(* IEC 61131-3 sources: TA/Tests/RetainTest/OLD/Structure test (part 9) *)

(* ---- StructureArrayTest.st ---- *)
PROGRAM StructureArrayTest

// СТРУКТУРА МАССИВОВ
IF TRIGGER_IMP.Q THEN

    ARRAY_STRUCTURE_RETAIN.ARRAY_BOOL[0] := NOT ARRAY_STRUCTURE_RETAIN.ARRAY_BOOL[0];
    ARRAY_STRUCTURE_RETAIN.ARRAY_BOOL[1] := NOT ARRAY_STRUCTURE_RETAIN.ARRAY_BOOL[1];
    ARRAY_STRUCTURE_RETAIN.ARRAY_BOOL[2] := NOT ARRAY_STRUCTURE_RETAIN.ARRAY_BOOL[2];
    ARRAY_STRUCTURE_RETAIN.ARRAY_BOOL[3] := NOT ARRAY_STRUCTURE_RETAIN.ARRAY_BOOL[3];
    ARRAY_STRUCTURE_RETAIN.ARRAY_BOOL[4] := NOT ARRAY_STRUCTURE_RETAIN.ARRAY_BOOL[4];
    ARRAY_STRUCTURE_RETAIN.ARRAY_BOOL[5] := NOT ARRAY_STRUCTURE_RETAIN.ARRAY_BOOL[5];
    ARRAY_STRUCTURE_RETAIN.ARRAY_BOOL[6] := NOT ARRAY_STRUCTURE_RETAIN.ARRAY_BOOL[6];
    ARRAY_STRUCTURE_RETAIN.ARRAY_BOOL[7] := NOT ARRAY_STRUCTURE_RETAIN.ARRAY_BOOL[7];
    ARRAY_STRUCTURE_RETAIN.ARRAY_BOOL[8] := ARRAY_STRUCTURE_RETAIN.ARRAY_BOOL[6];
    ARRAY_STRUCTURE_RETAIN.ARRAY_BOOL[9] := ARRAY_STRUCTURE_RETAIN.ARRAY_BOOL[7];

    ARRAY_STRUCTURE_RETAIN.ARRAY_BYTE[0] := ARRAY_STRUCTURE_RETAIN.ARRAY_BYTE[0] + 1;
    ARRAY_STRUCTURE_RETAIN.ARRAY_BYTE[1] := ARRAY_STRUCTURE_RETAIN.ARRAY_BYTE[1] + 1;
    ARRAY_STRUCTURE_RETAIN.ARRAY_BYTE[2] := ARRAY_STRUCTURE_RETAIN.ARRAY_BYTE[2] + 1;
    ARRAY_STRUCTURE_RETAIN.ARRAY_BYTE[3] := ARRAY_STRUCTURE_RETAIN.ARRAY_BYTE[3] + 1;
    ARRAY_STRUCTURE_RETAIN.ARRAY_BYTE[4] := ARRAY_STRUCTURE_RETAIN.ARRAY_BYTE[4] + 1;
    ARRAY_STRUCTURE_RETAIN.ARRAY_BYTE[5] := ARRAY_STRUCTURE_RETAIN.ARRAY_BYTE[5] + 1;
    ARRAY_STRUCTURE_RETAIN.ARRAY_BYTE[6] := ARRAY_STRUCTURE_RETAIN.ARRAY_BYTE[6] + 1;
    ARRAY_STRUCTURE_RETAIN.ARRAY_BYTE[7] := ARRAY_STRUCTURE_RETAIN.ARRAY_BYTE[7] + 1;
    ARRAY_STRUCTURE_RETAIN.ARRAY_BYTE[8] := ARRAY_STRUCTURE_RETAIN.ARRAY_BYTE[6];
    ARRAY_STRUCTURE_RETAIN.ARRAY_BYTE[9] := ARRAY_STRUCTURE_RETAIN.ARRAY_BYTE[7];

    ARRAY_STRUCTURE_RETAIN.ARRAY_DATE[0] := ANY_TO_DATE(1445385600 + ARRAY_STRUCTURE_RETAIN.ARRAY_DINT[0] * 86400);
    ARRAY_STRUCTURE_RETAIN.ARRAY_DATE[1] := ANY_TO_DATE(1445385600 + ARRAY_STRUCTURE_RETAIN.ARRAY_DINT[1] * 86400);
    ARRAY_STRUCTURE_RETAIN.ARRAY_DATE[2] := ANY_TO_DATE(1445385600 + ARRAY_STRUCTURE_RETAIN.ARRAY_DINT[2] * 86400);
    ARRAY_STRUCTURE_RETAIN.ARRAY_DATE[3] := ANY_TO_DATE(1445385600 + ARRAY_STRUCTURE_RETAIN.ARRAY_DINT[3] * 86400);
    ARRAY_STRUCTURE_RETAIN.ARRAY_DATE[4] := ANY_TO_DATE(1445385600 + ARRAY_STRUCTURE_RETAIN.ARRAY_DINT[4] * 86400);
    ARRAY_STRUCTURE_RETAIN.ARRAY_DATE[5] := ANY_TO_DATE(1445385600 + ARRAY_STRUCTURE_RETAIN.ARRAY_DINT[5] * 86400);
    ARRAY_STRUCTURE_RETAIN.ARRAY_DATE[6] := ANY_TO_DATE(1445385600 + ARRAY_STRUCTURE_RETAIN.ARRAY_DINT[6] * 86400);
    ARRAY_STRUCTURE_RETAIN.ARRAY_DATE[7] := ANY_TO_DATE(1445385600 + ARRAY_STRUCTURE_RETAIN.ARRAY_DINT[7] * 86400);
    ARRAY_STRUCTURE_RETAIN.ARRAY_DATE[8] := ARRAY_STRUCTURE_RETAIN.ARRAY_DATE[6];
    ARRAY_STRUCTURE_RETAIN.ARRAY_DATE[9] := ARRAY_STRUCTURE_RETAIN.ARRAY_DATE[7];

    ARRAY_STRUCTURE_RETAIN.ARRAY_DINT[0] := ARRAY_STRUCTURE_RETAIN.ARRAY_DINT[0] + 1;
    ARRAY_STRUCTURE_RETAIN.ARRAY_DINT[1] := ARRAY_STRUCTURE_RETAIN.ARRAY_DINT[1] + 1;
    ARRAY_STRUCTURE_RETAIN.ARRAY_DINT[2] := ARRAY_STRUCTURE_RETAIN.ARRAY_DINT[2] + 1;
    ARRAY_STRUCTURE_RETAIN.ARRAY_DINT[3] := ARRAY_STRUCTURE_RETAIN.ARRAY_DINT[3] + 1;
    ARRAY_STRUCTURE_RETAIN.ARRAY_DINT[4] := ARRAY_STRUCTURE_RETAIN.ARRAY_DINT[4] + 1;
    ARRAY_STRUCTURE_RETAIN.ARRAY_DINT[5] := ARRAY_STRUCTURE_RETAIN.ARRAY_DINT[5] + 1;
    ARRAY_STRUCTURE_RETAIN.ARRAY_DINT[6] := ARRAY_STRUCTURE_RETAIN.ARRAY_DINT[6] + 1;
    ARRAY_STRUCTURE_RETAIN.ARRAY_DINT[7] := ARRAY_STRUCTURE_RETAIN.ARRAY_DINT[7] + 1;
    ARRAY_STRUCTURE_RETAIN.ARRAY_DINT[8] := ARRAY_STRUCTURE_RETAIN.ARRAY_DINT[6];
    ARRAY_STRUCTURE_RETAIN.ARRAY_DINT[9] := ARRAY_STRUCTURE_RETAIN.ARRAY_DINT[7];

    ARRAY_STRUCTURE_RETAIN.ARRAY_DWORD[0] := ARRAY_STRUCTURE_RETAIN.ARRAY_DWORD[0] + 1;
    ARRAY_STRUCTURE_RETAIN.ARRAY_DWORD[1] := ARRAY_STRUCTURE_RETAIN.ARRAY_DWORD[1] + 1;
    ARRAY_STRUCTURE_RETAIN.ARRAY_DWORD[2] := ARRAY_STRUCTURE_RETAIN.ARRAY_DWORD[2] + 1;
    ARRAY_STRUCTURE_RETAIN.ARRAY_DWORD[3] := ARRAY_STRUCTURE_RETAIN.ARRAY_DWORD[3] + 1;
    ARRAY_STRUCTURE_RETAIN.ARRAY_DWORD[4] := ARRAY_STRUCTURE_RETAIN.ARRAY_DWORD[4] + 1;
    ARRAY_STRUCTURE_RETAIN.ARRAY_DWORD[5] := ARRAY_STRUCTURE_RETAIN.ARRAY_DWORD[5] + 1;
    ARRAY_STRUCTURE_RETAIN.ARRAY_DWORD[6] := ARRAY_STRUCTURE_RETAIN.ARRAY_DWORD[6] + 1;
    ARRAY_STRUCTURE_RETAIN.ARRAY_DWORD[7] := ARRAY_STRUCTURE_RETAIN.ARRAY_DWORD[7] + 1;
    ARRAY_STRUCTURE_RETAIN.ARRAY_DWORD[8] := ARRAY_STRUCTURE_RETAIN.ARRAY_DWORD[6];
    ARRAY_STRUCTURE_RETAIN.ARRAY_DWORD[9] := ARRAY_STRUCTURE_RETAIN.ARRAY_DWORD[7];

    ARRAY_STRUCTURE_RETAIN.ARRAY_INT[0] := ARRAY_STRUCTURE_RETAIN.ARRAY_INT[0] + 1;
    ARRAY_STRUCTURE_RETAIN.ARRAY_INT[1] := ARRAY_STRUCTURE_RETAIN.ARRAY_INT[1] + 1;
    ARRAY_STRUCTURE_RETAIN.ARRAY_INT[2] := ARRAY_STRUCTURE_RETAIN.ARRAY_INT[2] + 1;
    ARRAY_STRUCTURE_RETAIN.ARRAY_INT[3] := ARRAY_STRUCTURE_RETAIN.ARRAY_INT[3] + 1;
    ARRAY_STRUCTURE_RETAIN.ARRAY_INT[4] := ARRAY_STRUCTURE_RETAIN.ARRAY_INT[4] + 1;
    ARRAY_STRUCTURE_RETAIN.ARRAY_INT[5] := ARRAY_STRUCTURE_RETAIN.ARRAY_INT[5] + 1;
    ARRAY_STRUCTURE_RETAIN.ARRAY_INT[6] := ARRAY_STRUCTURE_RETAIN.ARRAY_INT[6] + 1;
    ARRAY_STRUCTURE_RETAIN.ARRAY_INT[7] := ARRAY_STRUCTURE_RETAIN.ARRAY_INT[7] + 1;
    ARRAY_STRUCTURE_RETAIN.ARRAY_INT[8] := ARRAY_STRUCTURE_RETAIN.ARRAY_INT[6];
    ARRAY_STRUCTURE_RETAIN.ARRAY_INT[9] := ARRAY_STRUCTURE_RETAIN.ARRAY_INT[7];

    ARRAY_STRUCTURE_RETAIN.ARRAY_LINT[0] := ARRAY_STRUCTURE_RETAIN.ARRAY_LINT[0] + 1;
    ARRAY_STRUCTURE_RETAIN.ARRAY_LINT[1] := ARRAY_STRUCTURE_RETAIN.ARRAY_LINT[1] + 1;
    ARRAY_STRUCTURE_RETAIN.ARRAY_LINT[2] := ARRAY_STRUCTURE_RETAIN.ARRAY_LINT[2] + 1;
    ARRAY_STRUCTURE_RETAIN.ARRAY_LINT[3] := ARRAY_STRUCTURE_RETAIN.ARRAY_LINT[3] + 1;
    ARRAY_STRUCTURE_RETAIN.ARRAY_LINT[4] := ARRAY_STRUCTURE_RETAIN.ARRAY_LINT[4] + 1;
    ARRAY_STRUCTURE_RETAIN.ARRAY_LINT[5] := ARRAY_STRUCTURE_RETAIN.ARRAY_LINT[5] + 1;
    ARRAY_STRUCTURE_RETAIN.ARRAY_LINT[6] := ARRAY_STRUCTURE_RETAIN.ARRAY_LINT[6] + 1;
    ARRAY_STRUCTURE_RETAIN.ARRAY_LINT[7] := ARRAY_STRUCTURE_RETAIN.ARRAY_LINT[7] + 1;
    ARRAY_STRUCTURE_RETAIN.ARRAY_LINT[8] := ARRAY_STRUCTURE_RETAIN.ARRAY_LINT[6];
    ARRAY_STRUCTURE_RETAIN.ARRAY_LINT[9] := ARRAY_STRUCTURE_RETAIN.ARRAY_LINT[7];

    ARRAY_STRUCTURE_RETAIN.ARRAY_LREAL[0] := ARRAY_STRUCTURE_RETAIN.ARRAY_LREAL[0] + 1;
    ARRAY_STRUCTURE_RETAIN.ARRAY_LREAL[1] := ARRAY_STRUCTURE_RETAIN.ARRAY_LREAL[1] + 1;
    ARRAY_STRUCTURE_RETAIN.ARRAY_LREAL[2] := ARRAY_STRUCTURE_RETAIN.ARRAY_LREAL[2] + 1;
    ARRAY_STRUCTURE_RETAIN.ARRAY_LREAL[3] := ARRAY_STRUCTURE_RETAIN.ARRAY_LREAL[3] + 1;
    ARRAY_STRUCTURE_RETAIN.ARRAY_LREAL[4] := ARRAY_STRUCTURE_RETAIN.ARRAY_LREAL[4] + 1;
    ARRAY_STRUCTURE_RETAIN.ARRAY_LREAL[5] := ARRAY_STRUCTURE_RETAIN.ARRAY_LREAL[5] + 1;
    ARRAY_STRUCTURE_RETAIN.ARRAY_LREAL[6] := ARRAY_STRUCTURE_RETAIN.ARRAY_LREAL[6] + 1;
    ARRAY_STRUCTURE_RETAIN.ARRAY_LREAL[7] := ARRAY_STRUCTURE_RETAIN.ARRAY_LREAL[7] + 1;
    ARRAY_STRUCTURE_RETAIN.ARRAY_LREAL[8] := ARRAY_STRUCTURE_RETAIN.ARRAY_LREAL[6];
    ARRAY_STRUCTURE_RETAIN.ARRAY_LREAL[9] := ARRAY_STRUCTURE_RETAIN.ARRAY_LREAL[7];

    ARRAY_STRUCTURE_RETAIN.ARRAY_LWORD[0] := ARRAY_STRUCTURE_RETAIN.ARRAY_LWORD[0] + 1;
    ARRAY_STRUCTURE_RETAIN.ARRAY_LWORD[1] := ARRAY_STRUCTURE_RETAIN.ARRAY_LWORD[1] + 1;
    ARRAY_STRUCTURE_RETAIN.ARRAY_LWORD[2] := ARRAY_STRUCTURE_RETAIN.ARRAY_LWORD[2] + 1;
    ARRAY_STRUCTURE_RETAIN.ARRAY_LWORD[3] := ARRAY_STRUCTURE_RETAIN.ARRAY_LWORD[3] + 1;
    ARRAY_STRUCTURE_RETAIN.ARRAY_LWORD[4] := ARRAY_STRUCTURE_RETAIN.ARRAY_LWORD[4] + 1;
    ARRAY_STRUCTURE_RETAIN.ARRAY_LWORD[5] := ARRAY_STRUCTURE_RETAIN.ARRAY_LWORD[5] + 1;
    ARRAY_STRUCTURE_RETAIN.ARRAY_LWORD[6] := ARRAY_STRUCTURE_RETAIN.ARRAY_LWORD[6] + 1;
    ARRAY_STRUCTURE_RETAIN.ARRAY_LWORD[7] := ARRAY_STRUCTURE_RETAIN.ARRAY_LWORD[7] + 1;
    ARRAY_STRUCTURE_RETAIN.ARRAY_LWORD[8] := ARRAY_STRUCTURE_RETAIN.ARRAY_LWORD[6];
    ARRAY_STRUCTURE_RETAIN.ARRAY_LWORD[9] := ARRAY_STRUCTURE_RETAIN.ARRAY_LWORD[7];

    ARRAY_STRUCTURE_RETAIN.ARRAY_REAL[0] := ARRAY_STRUCTURE_RETAIN.ARRAY_REAL[0] + 1;
    ARRAY_STRUCTURE_RETAIN.ARRAY_REAL[1] := ARRAY_STRUCTURE_RETAIN.ARRAY_REAL[1] + 1;
    ARRAY_STRUCTURE_RETAIN.ARRAY_REAL[2] := ARRAY_STRUCTURE_RETAIN.ARRAY_REAL[2] + 1;
    ARRAY_STRUCTURE_RETAIN.ARRAY_REAL[3] := ARRAY_STRUCTURE_RETAIN.ARRAY_REAL[3] + 1;
    ARRAY_STRUCTURE_RETAIN.ARRAY_REAL[4] := ARRAY_STRUCTURE_RETAIN.ARRAY_REAL[4] + 1;
    ARRAY_STRUCTURE_RETAIN.ARRAY_REAL[5] := ARRAY_STRUCTURE_RETAIN.ARRAY_REAL[5] + 1;
    ARRAY_STRUCTURE_RETAIN.ARRAY_REAL[6] := ARRAY_STRUCTURE_RETAIN.ARRAY_REAL[6] + 1;
    ARRAY_STRUCTURE_RETAIN.ARRAY_REAL[7] := ARRAY_STRUCTURE_RETAIN.ARRAY_REAL[7] + 1;
    ARRAY_STRUCTURE_RETAIN.ARRAY_REAL[8] := ARRAY_STRUCTURE_RETAIN.ARRAY_REAL[6];
    ARRAY_STRUCTURE_RETAIN.ARRAY_REAL[9] := ARRAY_STRUCTURE_RETAIN.ARRAY_REAL[7];

    ARRAY_STRUCTURE_RETAIN.ARRAY_SINT[0] := ARRAY_STRUCTURE_RETAIN.ARRAY_SINT[0] + 1;
    ARRAY_STRUCTURE_RETAIN.ARRAY_SINT[1] := ARRAY_STRUCTURE_RETAIN.ARRAY_SINT[1] + 1;
    ARRAY_STRUCTURE_RETAIN.ARRAY_SINT[2] := ARRAY_STRUCTURE_RETAIN.ARRAY_SINT[2] + 1;
    ARRAY_STRUCTURE_RETAIN.ARRAY_SINT[3] := ARRAY_STRUCTURE_RETAIN.ARRAY_SINT[3] + 1;
    ARRAY_STRUCTURE_RETAIN.ARRAY_SINT[4] := ARRAY_STRUCTURE_RETAIN.ARRAY_SINT[4] + 1;
    ARRAY_STRUCTURE_RETAIN.ARRAY_SINT[5] := ARRAY_STRUCTURE_RETAIN.ARRAY_SINT[5] + 1;
    ARRAY_STRUCTURE_RETAIN.ARRAY_SINT[6] := ARRAY_STRUCTURE_RETAIN.ARRAY_SINT[6] + 1;
    ARRAY_STRUCTURE_RETAIN.ARRAY_SINT[7] := ARRAY_STRUCTURE_RETAIN.ARRAY_SINT[7] + 1;
    ARRAY_STRUCTURE_RETAIN.ARRAY_SINT[8] := ARRAY_STRUCTURE_RETAIN.ARRAY_SINT[6];
    ARRAY_STRUCTURE_RETAIN.ARRAY_SINT[9] := ARRAY_STRUCTURE_RETAIN.ARRAY_SINT[7];

    ARRAY_STRUCTURE_RETAIN.ARRAY_STRING[0] := ANY_TO_STRING(ARRAY_STRUCTURE_RETAIN.ARRAY_DINT[0]) + ' ' + ANY_TO_STRING(ARRAY_STRUCTURE_RETAIN.ARRAY_TIME[0]);
    ARRAY_STRUCTURE_RETAIN.ARRAY_STRING[1] := ANY_TO_STRING(ARRAY_STRUCTURE_RETAIN.ARRAY_DINT[1]) + ' ' + ANY_TO_STRING(ARRAY_STRUCTURE_RETAIN.ARRAY_TIME[1]);
    ARRAY_STRUCTURE_RETAIN.ARRAY_STRING[2] := ANY_TO_STRING(ARRAY_STRUCTURE_RETAIN.ARRAY_DINT[2]) + ' ' + ANY_TO_STRING(ARRAY_STRUCTURE_RETAIN.ARRAY_TIME[2]);
    ARRAY_STRUCTURE_RETAIN.ARRAY_STRING[3] := ANY_TO_STRING(ARRAY_STRUCTURE_RETAIN.ARRAY_DINT[3]) + ' ' + ANY_TO_STRING(ARRAY_STRUCTURE_RETAIN.ARRAY_TIME[3]);
    ARRAY_STRUCTURE_RETAIN.ARRAY_STRING[4] := ANY_TO_STRING(ARRAY_STRUCTURE_RETAIN.ARRAY_DINT[4]) + ' ' + ANY_TO_STRING(ARRAY_STRUCTURE_RETAIN.ARRAY_TIME[4]);
    ARRAY_STRUCTURE_RETAIN.ARRAY_STRING[5] := ANY_TO_STRING(ARRAY_STRUCTURE_RETAIN.ARRAY_DINT[5]) + ' ' + ANY_TO_STRING(ARRAY_STRUCTURE_RETAIN.ARRAY_TIME[5]);
    ARRAY_STRUCTURE_RETAIN.ARRAY_STRING[6] := ANY_TO_STRING(ARRAY_STRUCTURE_RETAIN.ARRAY_DINT[6]) + ' ' + ANY_TO_STRING(ARRAY_STRUCTURE_RETAIN.ARRAY_TIME[6]);
    ARRAY_STRUCTURE_RETAIN.ARRAY_STRING[7] := ANY_TO_STRING(ARRAY_STRUCTURE_RETAIN.ARRAY_DINT[7]) + ' ' + ANY_TO_STRING(ARRAY_STRUCTURE_RETAIN.ARRAY_TIME[7]);
    ARRAY_STRUCTURE_RETAIN.ARRAY_STRING[8] := ARRAY_STRUCTURE_RETAIN.ARRAY_STRING[6];
    ARRAY_STRUCTURE_RETAIN.ARRAY_STRING[9] := ARRAY_STRUCTURE_RETAIN.ARRAY_STRING[7];

    ARRAY_STRUCTURE_RETAIN.ARRAY_TIME[0] := ARRAY_STRUCTURE_RETAIN.ARRAY_TIME[0] + PULSE_TIME;
    ARRAY_STRUCTURE_RETAIN.ARRAY_TIME[1] := ARRAY_STRUCTURE_RETAIN.ARRAY_TIME[1] + PULSE_TIME;
    ARRAY_STRUCTURE_RETAIN.ARRAY_TIME[2] := ARRAY_STRUCTURE_RETAIN.ARRAY_TIME[2] + PULSE_TIME;
    ARRAY_STRUCTURE_RETAIN.ARRAY_TIME[3] := ARRAY_STRUCTURE_RETAIN.ARRAY_TIME[3] + PULSE_TIME;
    ARRAY_STRUCTURE_RETAIN.ARRAY_TIME[4] := ARRAY_STRUCTURE_RETAIN.ARRAY_TIME[4] + PULSE_TIME;
    ARRAY_STRUCTURE_RETAIN.ARRAY_TIME[5] := ARRAY_STRUCTURE_RETAIN.ARRAY_TIME[5] + PULSE_TIME;
    ARRAY_STRUCTURE_RETAIN.ARRAY_TIME[6] := ARRAY_STRUCTURE_RETAIN.ARRAY_TIME[6] + PULSE_TIME;
    ARRAY_STRUCTURE_RETAIN.ARRAY_TIME[7] := ARRAY_STRUCTURE_RETAIN.ARRAY_TIME[7] + PULSE_TIME;
    ARRAY_STRUCTURE_RETAIN.ARRAY_TIME[8] := ARRAY_STRUCTURE_RETAIN.ARRAY_TIME[6];
    ARRAY_STRUCTURE_RETAIN.ARRAY_TIME[9] := ARRAY_STRUCTURE_RETAIN.ARRAY_TIME[7];

    ARRAY_STRUCTURE_RETAIN.ARRAY_UDINT[0] := ARRAY_STRUCTURE_RETAIN.ARRAY_UDINT[0] + 1;
    ARRAY_STRUCTURE_RETAIN.ARRAY_UDINT[1] := ARRAY_STRUCTURE_RETAIN.ARRAY_UDINT[1] + 1;
    ARRAY_STRUCTURE_RETAIN.ARRAY_UDINT[2] := ARRAY_STRUCTURE_RETAIN.ARRAY_UDINT[2] + 1;
    ARRAY_STRUCTURE_RETAIN.ARRAY_UDINT[3] := ARRAY_STRUCTURE_RETAIN.ARRAY_UDINT[3] + 1;
    ARRAY_STRUCTURE_RETAIN.ARRAY_UDINT[4] := ARRAY_STRUCTURE_RETAIN.ARRAY_UDINT[4] + 1;
    ARRAY_STRUCTURE_RETAIN.ARRAY_UDINT[5] := ARRAY_STRUCTURE_RETAIN.ARRAY_UDINT[5] + 1;
    ARRAY_STRUCTURE_RETAIN.ARRAY_UDINT[6] := ARRAY_STRUCTURE_RETAIN.ARRAY_UDINT[6] + 1;
    ARRAY_STRUCTURE_RETAIN.ARRAY_UDINT[7] := ARRAY_STRUCTURE_RETAIN.ARRAY_UDINT[7] + 1;
    ARRAY_STRUCTURE_RETAIN.ARRAY_UDINT[8] := ARRAY_STRUCTURE_RETAIN.ARRAY_UDINT[6];
    ARRAY_STRUCTURE_RETAIN.ARRAY_UDINT[9] := ARRAY_STRUCTURE_RETAIN.ARRAY_UDINT[7];

    ARRAY_STRUCTURE_RETAIN.ARRAY_UINT[0] := ARRAY_STRUCTURE_RETAIN.ARRAY_UINT[0] + 1;
    ARRAY_STRUCTURE_RETAIN.ARRAY_UINT[1] := ARRAY_STRUCTURE_RETAIN.ARRAY_UINT[1] + 1;
    ARRAY_STRUCTURE_RETAIN.ARRAY_UINT[2] := ARRAY_STRUCTURE_RETAIN.ARRAY_UINT[2] + 1;
    ARRAY_STRUCTURE_RETAIN.ARRAY_UINT[3] := ARRAY_STRUCTURE_RETAIN.ARRAY_UINT[3] + 1;
    ARRAY_STRUCTURE_RETAIN.ARRAY_UINT[4] := ARRAY_STRUCTURE_RETAIN.ARRAY_UINT[4] + 1;
    ARRAY_STRUCTURE_RETAIN.ARRAY_UINT[5] := ARRAY_STRUCTURE_RETAIN.ARRAY_UINT[5] + 1;
    ARRAY_STRUCTURE_RETAIN.ARRAY_UINT[6] := ARRAY_STRUCTURE_RETAIN.ARRAY_UINT[6] + 1;
    ARRAY_STRUCTURE_RETAIN.ARRAY_UINT[7] := ARRAY_STRUCTURE_RETAIN.ARRAY_UINT[7] + 1;
    ARRAY_STRUCTURE_RETAIN.ARRAY_UINT[8] := ARRAY_STRUCTURE_RETAIN.ARRAY_UINT[6];
    ARRAY_STRUCTURE_RETAIN.ARRAY_UINT[9] := ARRAY_STRUCTURE_RETAIN.ARRAY_UINT[7];

    ARRAY_STRUCTURE_RETAIN.ARRAY_ULINT[0] := ARRAY_STRUCTURE_RETAIN.ARRAY_ULINT[0] + 1;
    ARRAY_STRUCTURE_RETAIN.ARRAY_ULINT[1] := ARRAY_STRUCTURE_RETAIN.ARRAY_ULINT[1] + 1;
    ARRAY_STRUCTURE_RETAIN.ARRAY_ULINT[2] := ARRAY_STRUCTURE_RETAIN.ARRAY_ULINT[2] + 1;
    ARRAY_STRUCTURE_RETAIN.ARRAY_ULINT[3] := ARRAY_STRUCTURE_RETAIN.ARRAY_ULINT[3] + 1;
    ARRAY_STRUCTURE_RETAIN.ARRAY_ULINT[4] := ARRAY_STRUCTURE_RETAIN.ARRAY_ULINT[4] + 1;
    ARRAY_STRUCTURE_RETAIN.ARRAY_ULINT[5] := ARRAY_STRUCTURE_RETAIN.ARRAY_ULINT[5] + 1;
    ARRAY_STRUCTURE_RETAIN.ARRAY_ULINT[6] := ARRAY_STRUCTURE_RETAIN.ARRAY_ULINT[6] + 1;
    ARRAY_STRUCTURE_RETAIN.ARRAY_ULINT[7] := ARRAY_STRUCTURE_RETAIN.ARRAY_ULINT[7] + 1;
    ARRAY_STRUCTURE_RETAIN.ARRAY_ULINT[8] := ARRAY_STRUCTURE_RETAIN.ARRAY_ULINT[6];
    ARRAY_STRUCTURE_RETAIN.ARRAY_ULINT[9] := ARRAY_STRUCTURE_RETAIN.ARRAY_ULINT[7];

    ARRAY_STRUCTURE_RETAIN.ARRAY_USINT[0] := ARRAY_STRUCTURE_RETAIN.ARRAY_USINT[0] + 1;
    ARRAY_STRUCTURE_RETAIN.ARRAY_USINT[1] := ARRAY_STRUCTURE_RETAIN.ARRAY_USINT[1] + 1;
    ARRAY_STRUCTURE_RETAIN.ARRAY_USINT[2] := ARRAY_STRUCTURE_RETAIN.ARRAY_USINT[2] + 1;
    ARRAY_STRUCTURE_RETAIN.ARRAY_USINT[3] := ARRAY_STRUCTURE_RETAIN.ARRAY_USINT[3] + 1;
    ARRAY_STRUCTURE_RETAIN.ARRAY_USINT[4] := ARRAY_STRUCTURE_RETAIN.ARRAY_USINT[4] + 1;
    ARRAY_STRUCTURE_RETAIN.ARRAY_USINT[5] := ARRAY_STRUCTURE_RETAIN.ARRAY_USINT[5] + 1;
    ARRAY_STRUCTURE_RETAIN.ARRAY_USINT[6] := ARRAY_STRUCTURE_RETAIN.ARRAY_USINT[6] + 1;
    ARRAY_STRUCTURE_RETAIN.ARRAY_USINT[7] := ARRAY_STRUCTURE_RETAIN.ARRAY_USINT[7] + 1;
    ARRAY_STRUCTURE_RETAIN.ARRAY_USINT[8] := ARRAY_STRUCTURE_RETAIN.ARRAY_USINT[6];
    ARRAY_STRUCTURE_RETAIN.ARRAY_USINT[9] := ARRAY_STRUCTURE_RETAIN.ARRAY_USINT[7];

    ARRAY_STRUCTURE_RETAIN.ARRAY_WORD[0] := ARRAY_STRUCTURE_RETAIN.ARRAY_WORD[0] + 1;
    ARRAY_STRUCTURE_RETAIN.ARRAY_WORD[1] := ARRAY_STRUCTURE_RETAIN.ARRAY_WORD[1] + 1;
    ARRAY_STRUCTURE_RETAIN.ARRAY_WORD[2] := ARRAY_STRUCTURE_RETAIN.ARRAY_WORD[2] + 1;
    ARRAY_STRUCTURE_RETAIN.ARRAY_WORD[3] := ARRAY_STRUCTURE_RETAIN.ARRAY_WORD[3] + 1;
    ARRAY_STRUCTURE_RETAIN.ARRAY_WORD[4] := ARRAY_STRUCTURE_RETAIN.ARRAY_WORD[4] + 1;
    ARRAY_STRUCTURE_RETAIN.ARRAY_WORD[5] := ARRAY_STRUCTURE_RETAIN.ARRAY_WORD[5] + 1;
    ARRAY_STRUCTURE_RETAIN.ARRAY_WORD[6] := ARRAY_STRUCTURE_RETAIN.ARRAY_WORD[6] + 1;
    ARRAY_STRUCTURE_RETAIN.ARRAY_WORD[7] := ARRAY_STRUCTURE_RETAIN.ARRAY_WORD[7] + 1;
    ARRAY_STRUCTURE_RETAIN.ARRAY_WORD[8] := ARRAY_STRUCTURE_RETAIN.ARRAY_WORD[6];
    ARRAY_STRUCTURE_RETAIN.ARRAY_WORD[9] := ARRAY_STRUCTURE_RETAIN.ARRAY_WORD[7];

    ARRAY_STRUCTURE_NON_RETAIN.ARRAY_BOOL[0] := NOT ARRAY_STRUCTURE_NON_RETAIN.ARRAY_BOOL[0];
    ARRAY_STRUCTURE_NON_RETAIN.ARRAY_BOOL[1] := NOT ARRAY_STRUCTURE_NON_RETAIN.ARRAY_BOOL[1];
    ARRAY_STRUCTURE_NON_RETAIN.ARRAY_BOOL[2] := NOT ARRAY_STRUCTURE_NON_RETAIN.ARRAY_BOOL[2];
    ARRAY_STRUCTURE_NON_RETAIN.ARRAY_BOOL[3] := NOT ARRAY_STRUCTURE_NON_RETAIN.ARRAY_BOOL[3];
    ARRAY_STRUCTURE_NON_RETAIN.ARRAY_BOOL[4] := NOT ARRAY_STRUCTURE_NON_RETAIN.ARRAY_BOOL[4];
    ARRAY_STRUCTURE_NON_RETAIN.ARRAY_BOOL[5] := NOT ARRAY_STRUCTURE_NON_RETAIN.ARRAY_BOOL[5];
    ARRAY_STRUCTURE_NON_RETAIN.ARRAY_BOOL[6] := NOT ARRAY_STRUCTURE_NON_RETAIN.ARRAY_BOOL[6];
    ARRAY_STRUCTURE_NON_RETAIN.ARRAY_BOOL[7] := NOT ARRAY_STRUCTURE_NON_RETAIN.ARRAY_BOOL[7];
    ARRAY_STRUCTURE_NON_RETAIN.ARRAY_BOOL[8] := ARRAY_STRUCTURE_NON_RETAIN.ARRAY_BOOL[6];
    ARRAY_STRUCTURE_NON_RETAIN.ARRAY_BOOL[9] := ARRAY_STRUCTURE_NON_RETAIN.ARRAY_BOOL[7];

    ARRAY_STRUCTURE_NON_RETAIN.ARRAY_BYTE[0] := ARRAY_STRUCTURE_NON_RETAIN.ARRAY_BYTE[0] + 1;
    ARRAY_STRUCTURE_NON_RETAIN.ARRAY_BYTE[1] := ARRAY_STRUCTURE_NON_RETAIN.ARRAY_BYTE[1] + 1;
    ARRAY_STRUCTURE_NON_RETAIN.ARRAY_BYTE[2] := ARRAY_STRUCTURE_NON_RETAIN.ARRAY_BYTE[2] + 1;
    ARRAY_STRUCTURE_NON_RETAIN.ARRAY_BYTE[3] := ARRAY_STRUCTURE_NON_RETAIN.ARRAY_BYTE[3] + 1;
    ARRAY_STRUCTURE_NON_RETAIN.ARRAY_BYTE[4] := ARRAY_STRUCTURE_NON_RETAIN.ARRAY_BYTE[4] + 1;
    ARRAY_STRUCTURE_NON_RETAIN.ARRAY_BYTE[5] := ARRAY_STRUCTURE_NON_RETAIN.ARRAY_BYTE[5] + 1;
    ARRAY_STRUCTURE_NON_RETAIN.ARRAY_BYTE[6] := ARRAY_STRUCTURE_NON_RETAIN.ARRAY_BYTE[6] + 1;
    ARRAY_STRUCTURE_NON_RETAIN.ARRAY_BYTE[7] := ARRAY_STRUCTURE_NON_RETAIN.ARRAY_BYTE[7] + 1;
    ARRAY_STRUCTURE_NON_RETAIN.ARRAY_BYTE[8] := ARRAY_STRUCTURE_NON_RETAIN.ARRAY_BYTE[6];
    ARRAY_STRUCTURE_NON_RETAIN.ARRAY_BYTE[9] := ARRAY_STRUCTURE_NON_RETAIN.ARRAY_BYTE[7];

    ARRAY_STRUCTURE_NON_RETAIN.ARRAY_DATE[0] := ANY_TO_DATE(1445385600 + ARRAY_STRUCTURE_NON_RETAIN.ARRAY_DINT[0] * 86400);
    ARRAY_STRUCTURE_NON_RETAIN.ARRAY_DATE[1] := ANY_TO_DATE(1445385600 + ARRAY_STRUCTURE_NON_RETAIN.ARRAY_DINT[1] * 86400);
    ARRAY_STRUCTURE_NON_RETAIN.ARRAY_DATE[2] := ANY_TO_DATE(1445385600 + ARRAY_STRUCTURE_NON_RETAIN.ARRAY_DINT[2] * 86400);
    ARRAY_STRUCTURE_NON_RETAIN.ARRAY_DATE[3] := ANY_TO_DATE(1445385600 + ARRAY_STRUCTURE_NON_RETAIN.ARRAY_DINT[3] * 86400);
    ARRAY_STRUCTURE_NON_RETAIN.ARRAY_DATE[4] := ANY_TO_DATE(1445385600 + ARRAY_STRUCTURE_NON_RETAIN.ARRAY_DINT[4] * 86400);
    ARRAY_STRUCTURE_NON_RETAIN.ARRAY_DATE[5] := ANY_TO_DATE(1445385600 + ARRAY_STRUCTURE_NON_RETAIN.ARRAY_DINT[5] * 86400);
    ARRAY_STRUCTURE_NON_RETAIN.ARRAY_DATE[6] := ANY_TO_DATE(1445385600 + ARRAY_STRUCTURE_NON_RETAIN.ARRAY_DINT[6] * 86400);
    ARRAY_STRUCTURE_NON_RETAIN.ARRAY_DATE[7] := ANY_TO_DATE(1445385600 + ARRAY_STRUCTURE_NON_RETAIN.ARRAY_DINT[7] * 86400);
    ARRAY_STRUCTURE_NON_RETAIN.ARRAY_DATE[8] := ARRAY_STRUCTURE_NON_RETAIN.ARRAY_DATE[6];
    ARRAY_STRUCTURE_NON_RETAIN.ARRAY_DATE[9] := ARRAY_STRUCTURE_NON_RETAIN.ARRAY_DATE[7];

    ARRAY_STRUCTURE_NON_RETAIN.ARRAY_DINT[0] := ARRAY_STRUCTURE_NON_RETAIN.ARRAY_DINT[0] + 1;
    ARRAY_STRUCTURE_NON_RETAIN.ARRAY_DINT[1] := ARRAY_STRUCTURE_NON_RETAIN.ARRAY_DINT[1] + 1;
    ARRAY_STRUCTURE_NON_RETAIN.ARRAY_DINT[2] := ARRAY_STRUCTURE_NON_RETAIN.ARRAY_DINT[2] + 1;
    ARRAY_STRUCTURE_NON_RETAIN.ARRAY_DINT[3] := ARRAY_STRUCTURE_NON_RETAIN.ARRAY_DINT[3] + 1;
    ARRAY_STRUCTURE_NON_RETAIN.ARRAY_DINT[4] := ARRAY_STRUCTURE_NON_RETAIN.ARRAY_DINT[4] + 1;
    ARRAY_STRUCTURE_NON_RETAIN.ARRAY_DINT[5] := ARRAY_STRUCTURE_NON_RETAIN.ARRAY_DINT[5] + 1;
    ARRAY_STRUCTURE_NON_RETAIN.ARRAY_DINT[6] := ARRAY_STRUCTURE_NON_RETAIN.ARRAY_DINT[6] + 1;
    ARRAY_STRUCTURE_NON_RETAIN.ARRAY_DINT[7] := ARRAY_STRUCTURE_NON_RETAIN.ARRAY_DINT[7] + 1;
    ARRAY_STRUCTURE_NON_RETAIN.ARRAY_DINT[8] := ARRAY_STRUCTURE_NON_RETAIN.ARRAY_DINT[6];
    ARRAY_STRUCTURE_NON_RETAIN.ARRAY_DINT[9] := ARRAY_STRUCTURE_NON_RETAIN.ARRAY_DINT[7];

    ARRAY_STRUCTURE_NON_RETAIN.ARRAY_DWORD[0] := ARRAY_STRUCTURE_NON_RETAIN.ARRAY_DWORD[0] + 1;
    ARRAY_STRUCTURE_NON_RETAIN.ARRAY_DWORD[1] := ARRAY_STRUCTURE_NON_RETAIN.ARRAY_DWORD[1] + 1;
    ARRAY_STRUCTURE_NON_RETAIN.ARRAY_DWORD[2] := ARRAY_STRUCTURE_NON_RETAIN.ARRAY_DWORD[2] + 1;
    ARRAY_STRUCTURE_NON_RETAIN.ARRAY_DWORD[3] := ARRAY_STRUCTURE_NON_RETAIN.ARRAY_DWORD[3] + 1;
    ARRAY_STRUCTURE_NON_RETAIN.ARRAY_DWORD[4] := ARRAY_STRUCTURE_NON_RETAIN.ARRAY_DWORD[4] + 1;
    ARRAY_STRUCTURE_NON_RETAIN.ARRAY_DWORD[5] := ARRAY_STRUCTURE_NON_RETAIN.ARRAY_DWORD[5] + 1;
    ARRAY_STRUCTURE_NON_RETAIN.ARRAY_DWORD[6] := ARRAY_STRUCTURE_NON_RETAIN.ARRAY_DWORD[6] + 1;
    ARRAY_STRUCTURE_NON_RETAIN.ARRAY_DWORD[7] := ARRAY_STRUCTURE_NON_RETAIN.ARRAY_DWORD[7] + 1;
    ARRAY_STRUCTURE_NON_RETAIN.ARRAY_DWORD[8] := ARRAY_STRUCTURE_NON_RETAIN.ARRAY_DWORD[6];
    ARRAY_STRUCTURE_NON_RETAIN.ARRAY_DWORD[9] := ARRAY_STRUCTURE_NON_RETAIN.ARRAY_DWORD[7];

    ARRAY_STRUCTURE_NON_RETAIN.ARRAY_INT[0] := ARRAY_STRUCTURE_NON_RETAIN.ARRAY_INT[0] + 1;
    ARRAY_STRUCTURE_NON_RETAIN.ARRAY_INT[1] := ARRAY_STRUCTURE_NON_RETAIN.ARRAY_INT[1] + 1;
    ARRAY_STRUCTURE_NON_RETAIN.ARRAY_INT[2] := ARRAY_STRUCTURE_NON_RETAIN.ARRAY_INT[2] + 1;
    ARRAY_STRUCTURE_NON_RETAIN.ARRAY_INT[3] := ARRAY_STRUCTURE_NON_RETAIN.ARRAY_INT[3] + 1;
    ARRAY_STRUCTURE_NON_RETAIN.ARRAY_INT[4] := ARRAY_STRUCTURE_NON_RETAIN.ARRAY_INT[4] + 1;
    ARRAY_STRUCTURE_NON_RETAIN.ARRAY_INT[5] := ARRAY_STRUCTURE_NON_RETAIN.ARRAY_INT[5] + 1;
    ARRAY_STRUCTURE_NON_RETAIN.ARRAY_INT[6] := ARRAY_STRUCTURE_NON_RETAIN.ARRAY_INT[6] + 1;
    ARRAY_STRUCTURE_NON_RETAIN.ARRAY_INT[7] := ARRAY_STRUCTURE_NON_RETAIN.ARRAY_INT[7] + 1;
    ARRAY_STRUCTURE_NON_RETAIN.ARRAY_INT[8] := ARRAY_STRUCTURE_NON_RETAIN.ARRAY_INT[6];
    ARRAY_STRUCTURE_NON_RETAIN.ARRAY_INT[9] := ARRAY_STRUCTURE_NON_RETAIN.ARRAY_INT[7];

    ARRAY_STRUCTURE_NON_RETAIN.ARRAY_LINT[0] := ARRAY_STRUCTURE_NON_RETAIN.ARRAY_LINT[0] + 1;
    ARRAY_STRUCTURE_NON_RETAIN.ARRAY_LINT[1] := ARRAY_STRUCTURE_NON_RETAIN.ARRAY_LINT[1] + 1;
    ARRAY_STRUCTURE_NON_RETAIN.ARRAY_LINT[2] := ARRAY_STRUCTURE_NON_RETAIN.ARRAY_LINT[2] + 1;
    ARRAY_STRUCTURE_NON_RETAIN.ARRAY_LINT[3] := ARRAY_STRUCTURE_NON_RETAIN.ARRAY_LINT[3] + 1;
    ARRAY_STRUCTURE_NON_RETAIN.ARRAY_LINT[4] := ARRAY_STRUCTURE_NON_RETAIN.ARRAY_LINT[4] + 1;
    ARRAY_STRUCTURE_NON_RETAIN.ARRAY_LINT[5] := ARRAY_STRUCTURE_NON_RETAIN.ARRAY_LINT[5] + 1;
    ARRAY_STRUCTURE_NON_RETAIN.ARRAY_LINT[6] := ARRAY_STRUCTURE_NON_RETAIN.ARRAY_LINT[6] + 1;
    ARRAY_STRUCTURE_NON_RETAIN.ARRAY_LINT[7] := ARRAY_STRUCTURE_NON_RETAIN.ARRAY_LINT[7] + 1;
    ARRAY_STRUCTURE_NON_RETAIN.ARRAY_LINT[8] := ARRAY_STRUCTURE_NON_RETAIN.ARRAY_LINT[6];
    ARRAY_STRUCTURE_NON_RETAIN.ARRAY_LINT[9] := ARRAY_STRUCTURE_NON_RETAIN.ARRAY_LINT[7];

    ARRAY_STRUCTURE_NON_RETAIN.ARRAY_LREAL[0] := ARRAY_STRUCTURE_NON_RETAIN.ARRAY_LREAL[0] + 1;
    ARRAY_STRUCTURE_NON_RETAIN.ARRAY_LREAL[1] := ARRAY_STRUCTURE_NON_RETAIN.ARRAY_LREAL[1] + 1;
    ARRAY_STRUCTURE_NON_RETAIN.ARRAY_LREAL[2] := ARRAY_STRUCTURE_NON_RETAIN.ARRAY_LREAL[2] + 1;
    ARRAY_STRUCTURE_NON_RETAIN.ARRAY_LREAL[3] := ARRAY_STRUCTURE_NON_RETAIN.ARRAY_LREAL[3] + 1;
    ARRAY_STRUCTURE_NON_RETAIN.ARRAY_LREAL[4] := ARRAY_STRUCTURE_NON_RETAIN.ARRAY_LREAL[4] + 1;
    ARRAY_STRUCTURE_NON_RETAIN.ARRAY_LREAL[5] := ARRAY_STRUCTURE_NON_RETAIN.ARRAY_LREAL[5] + 1;
    ARRAY_STRUCTURE_NON_RETAIN.ARRAY_LREAL[6] := ARRAY_STRUCTURE_NON_RETAIN.ARRAY_LREAL[6] + 1;
    ARRAY_STRUCTURE_NON_RETAIN.ARRAY_LREAL[7] := ARRAY_STRUCTURE_NON_RETAIN.ARRAY_LREAL[7] + 1;
    ARRAY_STRUCTURE_NON_RETAIN.ARRAY_LREAL[8] := ARRAY_STRUCTURE_NON_RETAIN.ARRAY_LREAL[6];
    ARRAY_STRUCTURE_NON_RETAIN.ARRAY_LREAL[9] := ARRAY_STRUCTURE_NON_RETAIN.ARRAY_LREAL[7];

    ARRAY_STRUCTURE_NON_RETAIN.ARRAY_LWORD[0] := ARRAY_STRUCTURE_NON_RETAIN.ARRAY_LWORD[0] + 1;
    ARRAY_STRUCTURE_NON_RETAIN.ARRAY_LWORD[1] := ARRAY_STRUCTURE_NON_RETAIN.ARRAY_LWORD[1] + 1;
    ARRAY_STRUCTURE_NON_RETAIN.ARRAY_LWORD[2] := ARRAY_STRUCTURE_NON_RETAIN.ARRAY_LWORD[2] + 1;
    ARRAY_STRUCTURE_NON_RETAIN.ARRAY_LWORD[3] := ARRAY_STRUCTURE_NON_RETAIN.ARRAY_LWORD[3] + 1;
    ARRAY_STRUCTURE_NON_RETAIN.ARRAY_LWORD[4] := ARRAY_STRUCTURE_NON_RETAIN.ARRAY_LWORD[4] + 1;
    ARRAY_STRUCTURE_NON_RETAIN.ARRAY_LWORD[5] := ARRAY_STRUCTURE_NON_RETAIN.ARRAY_LWORD[5] + 1;
    ARRAY_STRUCTURE_NON_RETAIN.ARRAY_LWORD[6] := ARRAY_STRUCTURE_NON_RETAIN.ARRAY_LWORD[6] + 1;
    ARRAY_STRUCTURE_NON_RETAIN.ARRAY_LWORD[7] := ARRAY_STRUCTURE_NON_RETAIN.ARRAY_LWORD[7] + 1;
    ARRAY_STRUCTURE_NON_RETAIN.ARRAY_LWORD[8] := ARRAY_STRUCTURE_NON_RETAIN.ARRAY_LWORD[6];
    ARRAY_STRUCTURE_NON_RETAIN.ARRAY_LWORD[9] := ARRAY_STRUCTURE_NON_RETAIN.ARRAY_LWORD[7];

    ARRAY_STRUCTURE_NON_RETAIN.ARRAY_REAL[0] := ARRAY_STRUCTURE_NON_RETAIN.ARRAY_REAL[0] + 1;
    ARRAY_STRUCTURE_NON_RETAIN.ARRAY_REAL[1] := ARRAY_STRUCTURE_NON_RETAIN.ARRAY_REAL[1] + 1;
    ARRAY_STRUCTURE_NON_RETAIN.ARRAY_REAL[2] := ARRAY_STRUCTURE_NON_RETAIN.ARRAY_REAL[2] + 1;
    ARRAY_STRUCTURE_NON_RETAIN.ARRAY_REAL[3] := ARRAY_STRUCTURE_NON_RETAIN.ARRAY_REAL[3] + 1;
    ARRAY_STRUCTURE_NON_RETAIN.ARRAY_REAL[4] := ARRAY_STRUCTURE_NON_RETAIN.ARRAY_REAL[4] + 1;
    ARRAY_STRUCTURE_NON_RETAIN.ARRAY_REAL[5] := ARRAY_STRUCTURE_NON_RETAIN.ARRAY_REAL[5] + 1;
    ARRAY_STRUCTURE_NON_RETAIN.ARRAY_REAL[6] := ARRAY_STRUCTURE_NON_RETAIN.ARRAY_REAL[6] + 1;
    ARRAY_STRUCTURE_NON_RETAIN.ARRAY_REAL[7] := ARRAY_STRUCTURE_NON_RETAIN.ARRAY_REAL[7] + 1;
    ARRAY_STRUCTURE_NON_RETAIN.ARRAY_REAL[8] := ARRAY_STRUCTURE_NON_RETAIN.ARRAY_REAL[6];
    ARRAY_STRUCTURE_NON_RETAIN.ARRAY_REAL[9] := ARRAY_STRUCTURE_NON_RETAIN.ARRAY_REAL[7];

    ARRAY_STRUCTURE_NON_RETAIN.ARRAY_SINT[0] := ARRAY_STRUCTURE_NON_RETAIN.ARRAY_SINT[0] + 1;
    ARRAY_STRUCTURE_NON_RETAIN.ARRAY_SINT[1] := ARRAY_STRUCTURE_NON_RETAIN.ARRAY_SINT[1] + 1;
    ARRAY_STRUCTURE_NON_RETAIN.ARRAY_SINT[2] := ARRAY_STRUCTURE_NON_RETAIN.ARRAY_SINT[2] + 1;
    ARRAY_STRUCTURE_NON_RETAIN.ARRAY_SINT[3] := ARRAY_STRUCTURE_NON_RETAIN.ARRAY_SINT[3] + 1;
    ARRAY_STRUCTURE_NON_RETAIN.ARRAY_SINT[4] := ARRAY_STRUCTURE_NON_RETAIN.ARRAY_SINT[4] + 1;
    ARRAY_STRUCTURE_NON_RETAIN.ARRAY_SINT[5] := ARRAY_STRUCTURE_NON_RETAIN.ARRAY_SINT[5] + 1;
    ARRAY_STRUCTURE_NON_RETAIN.ARRAY_SINT[6] := ARRAY_STRUCTURE_NON_RETAIN.ARRAY_SINT[6] + 1;
    ARRAY_STRUCTURE_NON_RETAIN.ARRAY_SINT[7] := ARRAY_STRUCTURE_NON_RETAIN.ARRAY_SINT[7] + 1;
    ARRAY_STRUCTURE_NON_RETAIN.ARRAY_SINT[8] := ARRAY_STRUCTURE_NON_RETAIN.ARRAY_SINT[6];
    ARRAY_STRUCTURE_NON_RETAIN.ARRAY_SINT[9] := ARRAY_STRUCTURE_NON_RETAIN.ARRAY_SINT[7];

    ARRAY_STRUCTURE_NON_RETAIN.ARRAY_STRING[0] := ANY_TO_STRING(ARRAY_STRUCTURE_NON_RETAIN.ARRAY_DINT[0]) + ' ' + ANY_TO_STRING(ARRAY_STRUCTURE_NON_RETAIN.ARRAY_TIME[0]);
    ARRAY_STRUCTURE_NON_RETAIN.ARRAY_STRING[1] := ANY_TO_STRING(ARRAY_STRUCTURE_NON_RETAIN.ARRAY_DINT[1]) + ' ' + ANY_TO_STRING(ARRAY_STRUCTURE_NON_RETAIN.ARRAY_TIME[1]);
    ARRAY_STRUCTURE_NON_RETAIN.ARRAY_STRING[2] := ANY_TO_STRING(ARRAY_STRUCTURE_NON_RETAIN.ARRAY_DINT[2]) + ' ' + ANY_TO_STRING(ARRAY_STRUCTURE_NON_RETAIN.ARRAY_TIME[2]);
    ARRAY_STRUCTURE_NON_RETAIN.ARRAY_STRING[3] := ANY_TO_STRING(ARRAY_STRUCTURE_NON_RETAIN.ARRAY_DINT[3]) + ' ' + ANY_TO_STRING(ARRAY_STRUCTURE_NON_RETAIN.ARRAY_TIME[3]);
    ARRAY_STRUCTURE_NON_RETAIN.ARRAY_STRING[4] := ANY_TO_STRING(ARRAY_STRUCTURE_NON_RETAIN.ARRAY_DINT[4]) + ' ' + ANY_TO_STRING(ARRAY_STRUCTURE_NON_RETAIN.ARRAY_TIME[4]);
    ARRAY_STRUCTURE_NON_RETAIN.ARRAY_STRING[5] := ANY_TO_STRING(ARRAY_STRUCTURE_NON_RETAIN.ARRAY_DINT[5]) + ' ' + ANY_TO_STRING(ARRAY_STRUCTURE_NON_RETAIN.ARRAY_TIME[5]);
    ARRAY_STRUCTURE_NON_RETAIN.ARRAY_STRING[6] := ANY_TO_STRING(ARRAY_STRUCTURE_NON_RETAIN.ARRAY_DINT[6]) + ' ' + ANY_TO_STRING(ARRAY_STRUCTURE_NON_RETAIN.ARRAY_TIME[6]);
    ARRAY_STRUCTURE_NON_RETAIN.ARRAY_STRING[7] := ANY_TO_STRING(ARRAY_STRUCTURE_NON_RETAIN.ARRAY_DINT[7]) + ' ' + ANY_TO_STRING(ARRAY_STRUCTURE_NON_RETAIN.ARRAY_TIME[7]);
    ARRAY_STRUCTURE_NON_RETAIN.ARRAY_STRING[8] := ARRAY_STRUCTURE_NON_RETAIN.ARRAY_STRING[6];
    ARRAY_STRUCTURE_NON_RETAIN.ARRAY_STRING[9] := ARRAY_STRUCTURE_NON_RETAIN.ARRAY_STRING[7];

    ARRAY_STRUCTURE_NON_RETAIN.ARRAY_TIME[0] := ARRAY_STRUCTURE_NON_RETAIN.ARRAY_TIME[0] + PULSE_TIME;
    ARRAY_STRUCTURE_NON_RETAIN.ARRAY_TIME[1] := ARRAY_STRUCTURE_NON_RETAIN.ARRAY_TIME[1] + PULSE_TIME;
    ARRAY_STRUCTURE_NON_RETAIN.ARRAY_TIME[2] := ARRAY_STRUCTURE_NON_RETAIN.ARRAY_TIME[2] + PULSE_TIME;
    ARRAY_STRUCTURE_NON_RETAIN.ARRAY_TIME[3] := ARRAY_STRUCTURE_NON_RETAIN.ARRAY_TIME[3] + PULSE_TIME;
    ARRAY_STRUCTURE_NON_RETAIN.ARRAY_TIME[4] := ARRAY_STRUCTURE_NON_RETAIN.ARRAY_TIME[4] + PULSE_TIME;
    ARRAY_STRUCTURE_NON_RETAIN.ARRAY_TIME[5] := ARRAY_STRUCTURE_NON_RETAIN.ARRAY_TIME[5] + PULSE_TIME;
    ARRAY_STRUCTURE_NON_RETAIN.ARRAY_TIME[6] := ARRAY_STRUCTURE_NON_RETAIN.ARRAY_TIME[6] + PULSE_TIME;
    ARRAY_STRUCTURE_NON_RETAIN.ARRAY_TIME[7] := ARRAY_STRUCTURE_NON_RETAIN.ARRAY_TIME[7] + PULSE_TIME;
    ARRAY_STRUCTURE_NON_RETAIN.ARRAY_TIME[8] := ARRAY_STRUCTURE_NON_RETAIN.ARRAY_TIME[6];
    ARRAY_STRUCTURE_NON_RETAIN.ARRAY_TIME[9] := ARRAY_STRUCTURE_NON_RETAIN.ARRAY_TIME[7];

    ARRAY_STRUCTURE_NON_RETAIN.ARRAY_UDINT[0] := ARRAY_STRUCTURE_NON_RETAIN.ARRAY_UDINT[0] + 1;
    ARRAY_STRUCTURE_NON_RETAIN.ARRAY_UDINT[1] := ARRAY_STRUCTURE_NON_RETAIN.ARRAY_UDINT[1] + 1;
    ARRAY_STRUCTURE_NON_RETAIN.ARRAY_UDINT[2] := ARRAY_STRUCTURE_NON_RETAIN.ARRAY_UDINT[2] + 1;
    ARRAY_STRUCTURE_NON_RETAIN.ARRAY_UDINT[3] := ARRAY_STRUCTURE_NON_RETAIN.ARRAY_UDINT[3] + 1;
    ARRAY_STRUCTURE_NON_RETAIN.ARRAY_UDINT[4] := ARRAY_STRUCTURE_NON_RETAIN.ARRAY_UDINT[4] + 1;
    ARRAY_STRUCTURE_NON_RETAIN.ARRAY_UDINT[5] := ARRAY_STRUCTURE_NON_RETAIN.ARRAY_UDINT[5] + 1;
    ARRAY_STRUCTURE_NON_RETAIN.ARRAY_UDINT[6] := ARRAY_STRUCTURE_NON_RETAIN.ARRAY_UDINT[6] + 1;
    ARRAY_STRUCTURE_NON_RETAIN.ARRAY_UDINT[7] := ARRAY_STRUCTURE_NON_RETAIN.ARRAY_UDINT[7] + 1;
    ARRAY_STRUCTURE_NON_RETAIN.ARRAY_UDINT[8] := ARRAY_STRUCTURE_NON_RETAIN.ARRAY_UDINT[6];
    ARRAY_STRUCTURE_NON_RETAIN.ARRAY_UDINT[9] := ARRAY_STRUCTURE_NON_RETAIN.ARRAY_UDINT[7];

    ARRAY_STRUCTURE_NON_RETAIN.ARRAY_UINT[0] := ARRAY_STRUCTURE_NON_RETAIN.ARRAY_UINT[0] + 1;
    ARRAY_STRUCTURE_NON_RETAIN.ARRAY_UINT[1] := ARRAY_STRUCTURE_NON_RETAIN.ARRAY_UINT[1] + 1;
    ARRAY_STRUCTURE_NON_RETAIN.ARRAY_UINT[2] := ARRAY_STRUCTURE_NON_RETAIN.ARRAY_UINT[2] + 1;
    ARRAY_STRUCTURE_NON_RETAIN.ARRAY_UINT[3] := ARRAY_STRUCTURE_NON_RETAIN.ARRAY_UINT[3] + 1;
    ARRAY_STRUCTURE_NON_RETAIN.ARRAY_UINT[4] := ARRAY_STRUCTURE_NON_RETAIN.ARRAY_UINT[4] + 1;
    ARRAY_STRUCTURE_NON_RETAIN.ARRAY_UINT[5] := ARRAY_STRUCTURE_NON_RETAIN.ARRAY_UINT[5] + 1;
    ARRAY_STRUCTURE_NON_RETAIN.ARRAY_UINT[6] := ARRAY_STRUCTURE_NON_RETAIN.ARRAY_UINT[6] + 1;
    ARRAY_STRUCTURE_NON_RETAIN.ARRAY_UINT[7] := ARRAY_STRUCTURE_NON_RETAIN.ARRAY_UINT[7] + 1;
    ARRAY_STRUCTURE_NON_RETAIN.ARRAY_UINT[8] := ARRAY_STRUCTURE_NON_RETAIN.ARRAY_UINT[6];
    ARRAY_STRUCTURE_NON_RETAIN.ARRAY_UINT[9] := ARRAY_STRUCTURE_NON_RETAIN.ARRAY_UINT[7];

    ARRAY_STRUCTURE_NON_RETAIN.ARRAY_ULINT[0] := ARRAY_STRUCTURE_NON_RETAIN.ARRAY_ULINT[0] + 1;
    ARRAY_STRUCTURE_NON_RETAIN.ARRAY_ULINT[1] := ARRAY_STRUCTURE_NON_RETAIN.ARRAY_ULINT[1] + 1;
    ARRAY_STRUCTURE_NON_RETAIN.ARRAY_ULINT[2] := ARRAY_STRUCTURE_NON_RETAIN.ARRAY_ULINT[2] + 1;
    ARRAY_STRUCTURE_NON_RETAIN.ARRAY_ULINT[3] := ARRAY_STRUCTURE_NON_RETAIN.ARRAY_ULINT[3] + 1;
    ARRAY_STRUCTURE_NON_RETAIN.ARRAY_ULINT[4] := ARRAY_STRUCTURE_NON_RETAIN.ARRAY_ULINT[4] + 1;
    ARRAY_STRUCTURE_NON_RETAIN.ARRAY_ULINT[5] := ARRAY_STRUCTURE_NON_RETAIN.ARRAY_ULINT[5] + 1;
    ARRAY_STRUCTURE_NON_RETAIN.ARRAY_ULINT[6] := ARRAY_STRUCTURE_NON_RETAIN.ARRAY_ULINT[6] + 1;
    ARRAY_STRUCTURE_NON_RETAIN.ARRAY_ULINT[7] := ARRAY_STRUCTURE_NON_RETAIN.ARRAY_ULINT[7] + 1;
    ARRAY_STRUCTURE_NON_RETAIN.ARRAY_ULINT[8] := ARRAY_STRUCTURE_NON_RETAIN.ARRAY_ULINT[6];
    ARRAY_STRUCTURE_NON_RETAIN.ARRAY_ULINT[9] := ARRAY_STRUCTURE_NON_RETAIN.ARRAY_ULINT[7];

    ARRAY_STRUCTURE_NON_RETAIN.ARRAY_USINT[0] := ARRAY_STRUCTURE_NON_RETAIN.ARRAY_USINT[0] + 1;
    ARRAY_STRUCTURE_NON_RETAIN.ARRAY_USINT[1] := ARRAY_STRUCTURE_NON_RETAIN.ARRAY_USINT[1] + 1;
    ARRAY_STRUCTURE_NON_RETAIN.ARRAY_USINT[2] := ARRAY_STRUCTURE_NON_RETAIN.ARRAY_USINT[2] + 1;
    ARRAY_STRUCTURE_NON_RETAIN.ARRAY_USINT[3] := ARRAY_STRUCTURE_NON_RETAIN.ARRAY_USINT[3] + 1;
    ARRAY_STRUCTURE_NON_RETAIN.ARRAY_USINT[4] := ARRAY_STRUCTURE_NON_RETAIN.ARRAY_USINT[4] + 1;
    ARRAY_STRUCTURE_NON_RETAIN.ARRAY_USINT[5] := ARRAY_STRUCTURE_NON_RETAIN.ARRAY_USINT[5] + 1;
    ARRAY_STRUCTURE_NON_RETAIN.ARRAY_USINT[6] := ARRAY_STRUCTURE_NON_RETAIN.ARRAY_USINT[6] + 1;
    ARRAY_STRUCTURE_NON_RETAIN.ARRAY_USINT[7] := ARRAY_STRUCTURE_NON_RETAIN.ARRAY_USINT[7] + 1;
    ARRAY_STRUCTURE_NON_RETAIN.ARRAY_USINT[8] := ARRAY_STRUCTURE_NON_RETAIN.ARRAY_USINT[6];
    ARRAY_STRUCTURE_NON_RETAIN.ARRAY_USINT[9] := ARRAY_STRUCTURE_NON_RETAIN.ARRAY_USINT[7];

    ARRAY_STRUCTURE_NON_RETAIN.ARRAY_WORD[0] := ARRAY_STRUCTURE_NON_RETAIN.ARRAY_WORD[0] + 1;
    ARRAY_STRUCTURE_NON_RETAIN.ARRAY_WORD[1] := ARRAY_STRUCTURE_NON_RETAIN.ARRAY_WORD[1] + 1;
    ARRAY_STRUCTURE_NON_RETAIN.ARRAY_WORD[2] := ARRAY_STRUCTURE_NON_RETAIN.ARRAY_WORD[2] + 1;
    ARRAY_STRUCTURE_NON_RETAIN.ARRAY_WORD[3] := ARRAY_STRUCTURE_NON_RETAIN.ARRAY_WORD[3] + 1;
    ARRAY_STRUCTURE_NON_RETAIN.ARRAY_WORD[4] := ARRAY_STRUCTURE_NON_RETAIN.ARRAY_WORD[4] + 1;
    ARRAY_STRUCTURE_NON_RETAIN.ARRAY_WORD[5] := ARRAY_STRUCTURE_NON_RETAIN.ARRAY_WORD[5] + 1;
    ARRAY_STRUCTURE_NON_RETAIN.ARRAY_WORD[6] := ARRAY_STRUCTURE_NON_RETAIN.ARRAY_WORD[6] + 1;
    ARRAY_STRUCTURE_NON_RETAIN.ARRAY_WORD[7] := ARRAY_STRUCTURE_NON_RETAIN.ARRAY_WORD[7] + 1;
    ARRAY_STRUCTURE_NON_RETAIN.ARRAY_WORD[8] := ARRAY_STRUCTURE_NON_RETAIN.ARRAY_WORD[6];
    ARRAY_STRUCTURE_NON_RETAIN.ARRAY_WORD[9] := ARRAY_STRUCTURE_NON_RETAIN.ARRAY_WORD[7];

    ARRAY_STRUCTURE_AUTO.ARRAY_BOOL[0] := NOT ARRAY_STRUCTURE_AUTO.ARRAY_BOOL[0];
    ARRAY_STRUCTURE_AUTO.ARRAY_BOOL[1] := NOT ARRAY_STRUCTURE_AUTO.ARRAY_BOOL[1];
    ARRAY_STRUCTURE_AUTO.ARRAY_BOOL[2] := NOT ARRAY_STRUCTURE_AUTO.ARRAY_BOOL[2];
    ARRAY_STRUCTURE_AUTO.ARRAY_BOOL[3] := NOT ARRAY_STRUCTURE_AUTO.ARRAY_BOOL[3];
    ARRAY_STRUCTURE_AUTO.ARRAY_BOOL[4] := NOT ARRAY_STRUCTURE_AUTO.ARRAY_BOOL[4];
    ARRAY_STRUCTURE_AUTO.ARRAY_BOOL[5] := NOT ARRAY_STRUCTURE_AUTO.ARRAY_BOOL[5];
    ARRAY_STRUCTURE_AUTO.ARRAY_BOOL[6] := NOT ARRAY_STRUCTURE_AUTO.ARRAY_BOOL[6];
    ARRAY_STRUCTURE_AUTO.ARRAY_BOOL[7] := NOT ARRAY_STRUCTURE_AUTO.ARRAY_BOOL[7];
    ARRAY_STRUCTURE_AUTO.ARRAY_BOOL[8] := ARRAY_STRUCTURE_AUTO.ARRAY_BOOL[6];
    ARRAY_STRUCTURE_AUTO.ARRAY_BOOL[9] := ARRAY_STRUCTURE_AUTO.ARRAY_BOOL[7];

    ARRAY_STRUCTURE_AUTO.ARRAY_BYTE[0] := ARRAY_STRUCTURE_AUTO.ARRAY_BYTE[0] + 1;
    ARRAY_STRUCTURE_AUTO.ARRAY_BYTE[1] := ARRAY_STRUCTURE_AUTO.ARRAY_BYTE[1] + 1;
    ARRAY_STRUCTURE_AUTO.ARRAY_BYTE[2] := ARRAY_STRUCTURE_AUTO.ARRAY_BYTE[2] + 1;
    ARRAY_STRUCTURE_AUTO.ARRAY_BYTE[3] := ARRAY_STRUCTURE_AUTO.ARRAY_BYTE[3] + 1;
    ARRAY_STRUCTURE_AUTO.ARRAY_BYTE[4] := ARRAY_STRUCTURE_AUTO.ARRAY_BYTE[4] + 1;
    ARRAY_STRUCTURE_AUTO.ARRAY_BYTE[5] := ARRAY_STRUCTURE_AUTO.ARRAY_BYTE[5] + 1;
    ARRAY_STRUCTURE_AUTO.ARRAY_BYTE[6] := ARRAY_STRUCTURE_AUTO.ARRAY_BYTE[6] + 1;
    ARRAY_STRUCTURE_AUTO.ARRAY_BYTE[7] := ARRAY_STRUCTURE_AUTO.ARRAY_BYTE[7] + 1;
    ARRAY_STRUCTURE_AUTO.ARRAY_BYTE[8] := ARRAY_STRUCTURE_AUTO.ARRAY_BYTE[6];
    ARRAY_STRUCTURE_AUTO.ARRAY_BYTE[9] := ARRAY_STRUCTURE_AUTO.ARRAY_BYTE[7];

    ARRAY_STRUCTURE_AUTO.ARRAY_DATE[0] := ANY_TO_DATE(1445385600 + ARRAY_STRUCTURE_AUTO.ARRAY_DINT[0] * 86400);
    ARRAY_STRUCTURE_AUTO.ARRAY_DATE[1] := ANY_TO_DATE(1445385600 + ARRAY_STRUCTURE_AUTO.ARRAY_DINT[1] * 86400);
    ARRAY_STRUCTURE_AUTO.ARRAY_DATE[2] := ANY_TO_DATE(1445385600 + ARRAY_STRUCTURE_AUTO.ARRAY_DINT[2] * 86400);
    ARRAY_STRUCTURE_AUTO.ARRAY_DATE[3] := ANY_TO_DATE(1445385600 + ARRAY_STRUCTURE_AUTO.ARRAY_DINT[3] * 86400);
    ARRAY_STRUCTURE_AUTO.ARRAY_DATE[4] := ANY_TO_DATE(1445385600 + ARRAY_STRUCTURE_AUTO.ARRAY_DINT[4] * 86400);
    ARRAY_STRUCTURE_AUTO.ARRAY_DATE[5] := ANY_TO_DATE(1445385600 + ARRAY_STRUCTURE_AUTO.ARRAY_DINT[5] * 86400);
    ARRAY_STRUCTURE_AUTO.ARRAY_DATE[6] := ANY_TO_DATE(1445385600 + ARRAY_STRUCTURE_AUTO.ARRAY_DINT[6] * 86400);
    ARRAY_STRUCTURE_AUTO.ARRAY_DATE[7] := ANY_TO_DATE(1445385600 + ARRAY_STRUCTURE_AUTO.ARRAY_DINT[7] * 86400);
    ARRAY_STRUCTURE_AUTO.ARRAY_DATE[8] := ARRAY_STRUCTURE_AUTO.ARRAY_DATE[6];
    ARRAY_STRUCTURE_AUTO.ARRAY_DATE[9] := ARRAY_STRUCTURE_AUTO.ARRAY_DATE[7];

    ARRAY_STRUCTURE_AUTO.ARRAY_DINT[0] := ARRAY_STRUCTURE_AUTO.ARRAY_DINT[0] + 1;
    ARRAY_STRUCTURE_AUTO.ARRAY_DINT[1] := ARRAY_STRUCTURE_AUTO.ARRAY_DINT[1] + 1;
    ARRAY_STRUCTURE_AUTO.ARRAY_DINT[2] := ARRAY_STRUCTURE_AUTO.ARRAY_DINT[2] + 1;
    ARRAY_STRUCTURE_AUTO.ARRAY_DINT[3] := ARRAY_STRUCTURE_AUTO.ARRAY_DINT[3] + 1;
    ARRAY_STRUCTURE_AUTO.ARRAY_DINT[4] := ARRAY_STRUCTURE_AUTO.ARRAY_DINT[4] + 1;
    ARRAY_STRUCTURE_AUTO.ARRAY_DINT[5] := ARRAY_STRUCTURE_AUTO.ARRAY_DINT[5] + 1;
    ARRAY_STRUCTURE_AUTO.ARRAY_DINT[6] := ARRAY_STRUCTURE_AUTO.ARRAY_DINT[6] + 1;
    ARRAY_STRUCTURE_AUTO.ARRAY_DINT[7] := ARRAY_STRUCTURE_AUTO.ARRAY_DINT[7] + 1;
    ARRAY_STRUCTURE_AUTO.ARRAY_DINT[8] := ARRAY_STRUCTURE_AUTO.ARRAY_DINT[6];
    ARRAY_STRUCTURE_AUTO.ARRAY_DINT[9] := ARRAY_STRUCTURE_AUTO.ARRAY_DINT[7];

    ARRAY_STRUCTURE_AUTO.ARRAY_DWORD[0] := ARRAY_STRUCTURE_AUTO.ARRAY_DWORD[0] + 1;
    ARRAY_STRUCTURE_AUTO.ARRAY_DWORD[1] := ARRAY_STRUCTURE_AUTO.ARRAY_DWORD[1] + 1;
    ARRAY_STRUCTURE_AUTO.ARRAY_DWORD[2] := ARRAY_STRUCTURE_AUTO.ARRAY_DWORD[2] + 1;
    ARRAY_STRUCTURE_AUTO.ARRAY_DWORD[3] := ARRAY_STRUCTURE_AUTO.ARRAY_DWORD[3] + 1;
    ARRAY_STRUCTURE_AUTO.ARRAY_DWORD[4] := ARRAY_STRUCTURE_AUTO.ARRAY_DWORD[4] + 1;
    ARRAY_STRUCTURE_AUTO.ARRAY_DWORD[5] := ARRAY_STRUCTURE_AUTO.ARRAY_DWORD[5] + 1;
    ARRAY_STRUCTURE_AUTO.ARRAY_DWORD[6] := ARRAY_STRUCTURE_AUTO.ARRAY_DWORD[6] + 1;
    ARRAY_STRUCTURE_AUTO.ARRAY_DWORD[7] := ARRAY_STRUCTURE_AUTO.ARRAY_DWORD[7] + 1;
    ARRAY_STRUCTURE_AUTO.ARRAY_DWORD[8] := ARRAY_STRUCTURE_AUTO.ARRAY_DWORD[6];
    ARRAY_STRUCTURE_AUTO.ARRAY_DWORD[9] := ARRAY_STRUCTURE_AUTO.ARRAY_DWORD[7];

    ARRAY_STRUCTURE_AUTO.ARRAY_INT[0] := ARRAY_STRUCTURE_AUTO.ARRAY_INT[0] + 1;
    ARRAY_STRUCTURE_AUTO.ARRAY_INT[1] := ARRAY_STRUCTURE_AUTO.ARRAY_INT[1] + 1;
    ARRAY_STRUCTURE_AUTO.ARRAY_INT[2] := ARRAY_STRUCTURE_AUTO.ARRAY_INT[2] + 1;
    ARRAY_STRUCTURE_AUTO.ARRAY_INT[3] := ARRAY_STRUCTURE_AUTO.ARRAY_INT[3] + 1;
    ARRAY_STRUCTURE_AUTO.ARRAY_INT[4] := ARRAY_STRUCTURE_AUTO.ARRAY_INT[4] + 1;
    ARRAY_STRUCTURE_AUTO.ARRAY_INT[5] := ARRAY_STRUCTURE_AUTO.ARRAY_INT[5] + 1;
    ARRAY_STRUCTURE_AUTO.ARRAY_INT[6] := ARRAY_STRUCTURE_AUTO.ARRAY_INT[6] + 1;
    ARRAY_STRUCTURE_AUTO.ARRAY_INT[7] := ARRAY_STRUCTURE_AUTO.ARRAY_INT[7] + 1;
    ARRAY_STRUCTURE_AUTO.ARRAY_INT[8] := ARRAY_STRUCTURE_AUTO.ARRAY_INT[6];
    ARRAY_STRUCTURE_AUTO.ARRAY_INT[9] := ARRAY_STRUCTURE_AUTO.ARRAY_INT[7];

    ARRAY_STRUCTURE_AUTO.ARRAY_LINT[0] := ARRAY_STRUCTURE_AUTO.ARRAY_LINT[0] + 1;
    ARRAY_STRUCTURE_AUTO.ARRAY_LINT[1] := ARRAY_STRUCTURE_AUTO.ARRAY_LINT[1] + 1;
    ARRAY_STRUCTURE_AUTO.ARRAY_LINT[2] := ARRAY_STRUCTURE_AUTO.ARRAY_LINT[2] + 1;
    ARRAY_STRUCTURE_AUTO.ARRAY_LINT[3] := ARRAY_STRUCTURE_AUTO.ARRAY_LINT[3] + 1;
    ARRAY_STRUCTURE_AUTO.ARRAY_LINT[4] := ARRAY_STRUCTURE_AUTO.ARRAY_LINT[4] + 1;
    ARRAY_STRUCTURE_AUTO.ARRAY_LINT[5] := ARRAY_STRUCTURE_AUTO.ARRAY_LINT[5] + 1;
    ARRAY_STRUCTURE_AUTO.ARRAY_LINT[6] := ARRAY_STRUCTURE_AUTO.ARRAY_LINT[6] + 1;
    ARRAY_STRUCTURE_AUTO.ARRAY_LINT[7] := ARRAY_STRUCTURE_AUTO.ARRAY_LINT[7] + 1;
    ARRAY_STRUCTURE_AUTO.ARRAY_LINT[8] := ARRAY_STRUCTURE_AUTO.ARRAY_LINT[6];
    ARRAY_STRUCTURE_AUTO.ARRAY_LINT[9] := ARRAY_STRUCTURE_AUTO.ARRAY_LINT[7];

    ARRAY_STRUCTURE_AUTO.ARRAY_LREAL[0] := ARRAY_STRUCTURE_AUTO.ARRAY_LREAL[0] + 1;
    ARRAY_STRUCTURE_AUTO.ARRAY_LREAL[1] := ARRAY_STRUCTURE_AUTO.ARRAY_LREAL[1] + 1;
    ARRAY_STRUCTURE_AUTO.ARRAY_LREAL[2] := ARRAY_STRUCTURE_AUTO.ARRAY_LREAL[2] + 1;
    ARRAY_STRUCTURE_AUTO.ARRAY_LREAL[3] := ARRAY_STRUCTURE_AUTO.ARRAY_LREAL[3] + 1;
    ARRAY_STRUCTURE_AUTO.ARRAY_LREAL[4] := ARRAY_STRUCTURE_AUTO.ARRAY_LREAL[4] + 1;
    ARRAY_STRUCTURE_AUTO.ARRAY_LREAL[5] := ARRAY_STRUCTURE_AUTO.ARRAY_LREAL[5] + 1;
    ARRAY_STRUCTURE_AUTO.ARRAY_LREAL[6] := ARRAY_STRUCTURE_AUTO.ARRAY_LREAL[6] + 1;
    ARRAY_STRUCTURE_AUTO.ARRAY_LREAL[7] := ARRAY_STRUCTURE_AUTO.ARRAY_LREAL[7] + 1;
    ARRAY_STRUCTURE_AUTO.ARRAY_LREAL[8] := ARRAY_STRUCTURE_AUTO.ARRAY_LREAL[6];
    ARRAY_STRUCTURE_AUTO.ARRAY_LREAL[9] := ARRAY_STRUCTURE_AUTO.ARRAY_LREAL[7];

    ARRAY_STRUCTURE_AUTO.ARRAY_LWORD[0] := ARRAY_STRUCTURE_AUTO.ARRAY_LWORD[0] + 1;
    ARRAY_STRUCTURE_AUTO.ARRAY_LWORD[1] := ARRAY_STRUCTURE_AUTO.ARRAY_LWORD[1] + 1;
    ARRAY_STRUCTURE_AUTO.ARRAY_LWORD[2] := ARRAY_STRUCTURE_AUTO.ARRAY_LWORD[2] + 1;
    ARRAY_STRUCTURE_AUTO.ARRAY_LWORD[3] := ARRAY_STRUCTURE_AUTO.ARRAY_LWORD[3] + 1;
    ARRAY_STRUCTURE_AUTO.ARRAY_LWORD[4] := ARRAY_STRUCTURE_AUTO.ARRAY_LWORD[4] + 1;
    ARRAY_STRUCTURE_AUTO.ARRAY_LWORD[5] := ARRAY_STRUCTURE_AUTO.ARRAY_LWORD[5] + 1;
    ARRAY_STRUCTURE_AUTO.ARRAY_LWORD[6] := ARRAY_STRUCTURE_AUTO.ARRAY_LWORD[6] + 1;
    ARRAY_STRUCTURE_AUTO.ARRAY_LWORD[7] := ARRAY_STRUCTURE_AUTO.ARRAY_LWORD[7] + 1;
    ARRAY_STRUCTURE_AUTO.ARRAY_LWORD[8] := ARRAY_STRUCTURE_AUTO.ARRAY_LWORD[6];
    ARRAY_STRUCTURE_AUTO.ARRAY_LWORD[9] := ARRAY_STRUCTURE_AUTO.ARRAY_LWORD[7];

    ARRAY_STRUCTURE_AUTO.ARRAY_REAL[0] := ARRAY_STRUCTURE_AUTO.ARRAY_REAL[0] + 1;
    ARRAY_STRUCTURE_AUTO.ARRAY_REAL[1] := ARRAY_STRUCTURE_AUTO.ARRAY_REAL[1] + 1;
    ARRAY_STRUCTURE_AUTO.ARRAY_REAL[2] := ARRAY_STRUCTURE_AUTO.ARRAY_REAL[2] + 1;
    ARRAY_STRUCTURE_AUTO.ARRAY_REAL[3] := ARRAY_STRUCTURE_AUTO.ARRAY_REAL[3] + 1;
    ARRAY_STRUCTURE_AUTO.ARRAY_REAL[4] := ARRAY_STRUCTURE_AUTO.ARRAY_REAL[4] + 1;
    ARRAY_STRUCTURE_AUTO.ARRAY_REAL[5] := ARRAY_STRUCTURE_AUTO.ARRAY_REAL[5] + 1;
    ARRAY_STRUCTURE_AUTO.ARRAY_REAL[6] := ARRAY_STRUCTURE_AUTO.ARRAY_REAL[6] + 1;
    ARRAY_STRUCTURE_AUTO.ARRAY_REAL[7] := ARRAY_STRUCTURE_AUTO.ARRAY_REAL[7] + 1;
    ARRAY_STRUCTURE_AUTO.ARRAY_REAL[8] := ARRAY_STRUCTURE_AUTO.ARRAY_REAL[6];
    ARRAY_STRUCTURE_AUTO.ARRAY_REAL[9] := ARRAY_STRUCTURE_AUTO.ARRAY_REAL[7];

    ARRAY_STRUCTURE_AUTO.ARRAY_SINT[0] := ARRAY_STRUCTURE_AUTO.ARRAY_SINT[0] + 1;
    ARRAY_STRUCTURE_AUTO.ARRAY_SINT[1] := ARRAY_STRUCTURE_AUTO.ARRAY_SINT[1] + 1;
    ARRAY_STRUCTURE_AUTO.ARRAY_SINT[2] := ARRAY_STRUCTURE_AUTO.ARRAY_SINT[2] + 1;
    ARRAY_STRUCTURE_AUTO.ARRAY_SINT[3] := ARRAY_STRUCTURE_AUTO.ARRAY_SINT[3] + 1;
    ARRAY_STRUCTURE_AUTO.ARRAY_SINT[4] := ARRAY_STRUCTURE_AUTO.ARRAY_SINT[4] + 1;
    ARRAY_STRUCTURE_AUTO.ARRAY_SINT[5] := ARRAY_STRUCTURE_AUTO.ARRAY_SINT[5] + 1;
    ARRAY_STRUCTURE_AUTO.ARRAY_SINT[6] := ARRAY_STRUCTURE_AUTO.ARRAY_SINT[6] + 1;
    ARRAY_STRUCTURE_AUTO.ARRAY_SINT[7] := ARRAY_STRUCTURE_AUTO.ARRAY_SINT[7] + 1;
    ARRAY_STRUCTURE_AUTO.ARRAY_SINT[8] := ARRAY_STRUCTURE_AUTO.ARRAY_SINT[6];
    ARRAY_STRUCTURE_AUTO.ARRAY_SINT[9] := ARRAY_STRUCTURE_AUTO.ARRAY_SINT[7];

    ARRAY_STRUCTURE_AUTO.ARRAY_STRING[0] := ANY_TO_STRING(ARRAY_STRUCTURE_AUTO.ARRAY_DINT[0]) + ' ' + ANY_TO_STRING(ARRAY_STRUCTURE_AUTO.ARRAY_TIME[0]);
    ARRAY_STRUCTURE_AUTO.ARRAY_STRING[1] := ANY_TO_STRING(ARRAY_STRUCTURE_AUTO.ARRAY_DINT[1]) + ' ' + ANY_TO_STRING(ARRAY_STRUCTURE_AUTO.ARRAY_TIME[1]);
    ARRAY_STRUCTURE_AUTO.ARRAY_STRING[2] := ANY_TO_STRING(ARRAY_STRUCTURE_AUTO.ARRAY_DINT[2]) + ' ' + ANY_TO_STRING(ARRAY_STRUCTURE_AUTO.ARRAY_TIME[2]);
    ARRAY_STRUCTURE_AUTO.ARRAY_STRING[3] := ANY_TO_STRING(ARRAY_STRUCTURE_AUTO.ARRAY_DINT[3]) + ' ' + ANY_TO_STRING(ARRAY_STRUCTURE_AUTO.ARRAY_TIME[3]);
    ARRAY_STRUCTURE_AUTO.ARRAY_STRING[4] := ANY_TO_STRING(ARRAY_STRUCTURE_AUTO.ARRAY_DINT[4]) + ' ' + ANY_TO_STRING(ARRAY_STRUCTURE_AUTO.ARRAY_TIME[4]);
    ARRAY_STRUCTURE_AUTO.ARRAY_STRING[5] := ANY_TO_STRING(ARRAY_STRUCTURE_AUTO.ARRAY_DINT[5]) + ' ' + ANY_TO_STRING(ARRAY_STRUCTURE_AUTO.ARRAY_TIME[5]);
    ARRAY_STRUCTURE_AUTO.ARRAY_STRING[6] := ANY_TO_STRING(ARRAY_STRUCTURE_AUTO.ARRAY_DINT[6]) + ' ' + ANY_TO_STRING(ARRAY_STRUCTURE_AUTO.ARRAY_TIME[6]);
    ARRAY_STRUCTURE_AUTO.ARRAY_STRING[7] := ANY_TO_STRING(ARRAY_STRUCTURE_AUTO.ARRAY_DINT[7]) + ' ' + ANY_TO_STRING(ARRAY_STRUCTURE_AUTO.ARRAY_TIME[7]);
    ARRAY_STRUCTURE_AUTO.ARRAY_STRING[8] := ARRAY_STRUCTURE_AUTO.ARRAY_STRING[6];
    ARRAY_STRUCTURE_AUTO.ARRAY_STRING[9] := ARRAY_STRUCTURE_AUTO.ARRAY_STRING[7];

    ARRAY_STRUCTURE_AUTO.ARRAY_TIME[0] := ARRAY_STRUCTURE_AUTO.ARRAY_TIME[0] + PULSE_TIME;
    ARRAY_STRUCTURE_AUTO.ARRAY_TIME[1] := ARRAY_STRUCTURE_AUTO.ARRAY_TIME[1] + PULSE_TIME;
    ARRAY_STRUCTURE_AUTO.ARRAY_TIME[2] := ARRAY_STRUCTURE_AUTO.ARRAY_TIME[2] + PULSE_TIME;
    ARRAY_STRUCTURE_AUTO.ARRAY_TIME[3] := ARRAY_STRUCTURE_AUTO.ARRAY_TIME[3] + PULSE_TIME;
    ARRAY_STRUCTURE_AUTO.ARRAY_TIME[4] := ARRAY_STRUCTURE_AUTO.ARRAY_TIME[4] + PULSE_TIME;
    ARRAY_STRUCTURE_AUTO.ARRAY_TIME[5] := ARRAY_STRUCTURE_AUTO.ARRAY_TIME[5] + PULSE_TIME;
    ARRAY_STRUCTURE_AUTO.ARRAY_TIME[6] := ARRAY_STRUCTURE_AUTO.ARRAY_TIME[6] + PULSE_TIME;
    ARRAY_STRUCTURE_AUTO.ARRAY_TIME[7] := ARRAY_STRUCTURE_AUTO.ARRAY_TIME[7] + PULSE_TIME;
    ARRAY_STRUCTURE_AUTO.ARRAY_TIME[8] := ARRAY_STRUCTURE_AUTO.ARRAY_TIME[6];
    ARRAY_STRUCTURE_AUTO.ARRAY_TIME[9] := ARRAY_STRUCTURE_AUTO.ARRAY_TIME[7];

    ARRAY_STRUCTURE_AUTO.ARRAY_UDINT[0] := ARRAY_STRUCTURE_AUTO.ARRAY_UDINT[0] + 1;
    ARRAY_STRUCTURE_AUTO.ARRAY_UDINT[1] := ARRAY_STRUCTURE_AUTO.ARRAY_UDINT[1] + 1;
    ARRAY_STRUCTURE_AUTO.ARRAY_UDINT[2] := ARRAY_STRUCTURE_AUTO.ARRAY_UDINT[2] + 1;
    ARRAY_STRUCTURE_AUTO.ARRAY_UDINT[3] := ARRAY_STRUCTURE_AUTO.ARRAY_UDINT[3] + 1;
    ARRAY_STRUCTURE_AUTO.ARRAY_UDINT[4] := ARRAY_STRUCTURE_AUTO.ARRAY_UDINT[4] + 1;
    ARRAY_STRUCTURE_AUTO.ARRAY_UDINT[5] := ARRAY_STRUCTURE_AUTO.ARRAY_UDINT[5] + 1;
    ARRAY_STRUCTURE_AUTO.ARRAY_UDINT[6] := ARRAY_STRUCTURE_AUTO.ARRAY_UDINT[6] + 1;
    ARRAY_STRUCTURE_AUTO.ARRAY_UDINT[7] := ARRAY_STRUCTURE_AUTO.ARRAY_UDINT[7] + 1;
    ARRAY_STRUCTURE_AUTO.ARRAY_UDINT[8] := ARRAY_STRUCTURE_AUTO.ARRAY_UDINT[6];
    ARRAY_STRUCTURE_AUTO.ARRAY_UDINT[9] := ARRAY_STRUCTURE_AUTO.ARRAY_UDINT[7];

    ARRAY_STRUCTURE_AUTO.ARRAY_UINT[0] := ARRAY_STRUCTURE_AUTO.ARRAY_UINT[0] + 1;
    ARRAY_STRUCTURE_AUTO.ARRAY_UINT[1] := ARRAY_STRUCTURE_AUTO.ARRAY_UINT[1] + 1;
    ARRAY_STRUCTURE_AUTO.ARRAY_UINT[2] := ARRAY_STRUCTURE_AUTO.ARRAY_UINT[2] + 1;
    ARRAY_STRUCTURE_AUTO.ARRAY_UINT[3] := ARRAY_STRUCTURE_AUTO.ARRAY_UINT[3] + 1;
    ARRAY_STRUCTURE_AUTO.ARRAY_UINT[4] := ARRAY_STRUCTURE_AUTO.ARRAY_UINT[4] + 1;
    ARRAY_STRUCTURE_AUTO.ARRAY_UINT[5] := ARRAY_STRUCTURE_AUTO.ARRAY_UINT[5] + 1;
    ARRAY_STRUCTURE_AUTO.ARRAY_UINT[6] := ARRAY_STRUCTURE_AUTO.ARRAY_UINT[6] + 1;
    ARRAY_STRUCTURE_AUTO.ARRAY_UINT[7] := ARRAY_STRUCTURE_AUTO.ARRAY_UINT[7] + 1;
    ARRAY_STRUCTURE_AUTO.ARRAY_UINT[8] := ARRAY_STRUCTURE_AUTO.ARRAY_UINT[6];
    ARRAY_STRUCTURE_AUTO.ARRAY_UINT[9] := ARRAY_STRUCTURE_AUTO.ARRAY_UINT[7];

    ARRAY_STRUCTURE_AUTO.ARRAY_ULINT[0] := ARRAY_STRUCTURE_AUTO.ARRAY_ULINT[0] + 1;
    ARRAY_STRUCTURE_AUTO.ARRAY_ULINT[1] := ARRAY_STRUCTURE_AUTO.ARRAY_ULINT[1] + 1;
    ARRAY_STRUCTURE_AUTO.ARRAY_ULINT[2] := ARRAY_STRUCTURE_AUTO.ARRAY_ULINT[2] + 1;
    ARRAY_STRUCTURE_AUTO.ARRAY_ULINT[3] := ARRAY_STRUCTURE_AUTO.ARRAY_ULINT[3] + 1;
    ARRAY_STRUCTURE_AUTO.ARRAY_ULINT[4] := ARRAY_STRUCTURE_AUTO.ARRAY_ULINT[4] + 1;
    ARRAY_STRUCTURE_AUTO.ARRAY_ULINT[5] := ARRAY_STRUCTURE_AUTO.ARRAY_ULINT[5] + 1;
    ARRAY_STRUCTURE_AUTO.ARRAY_ULINT[6] := ARRAY_STRUCTURE_AUTO.ARRAY_ULINT[6] + 1;
    ARRAY_STRUCTURE_AUTO.ARRAY_ULINT[7] := ARRAY_STRUCTURE_AUTO.ARRAY_ULINT[7] + 1;
    ARRAY_STRUCTURE_AUTO.ARRAY_ULINT[8] := ARRAY_STRUCTURE_AUTO.ARRAY_ULINT[6];
    ARRAY_STRUCTURE_AUTO.ARRAY_ULINT[9] := ARRAY_STRUCTURE_AUTO.ARRAY_ULINT[7];

    ARRAY_STRUCTURE_AUTO.ARRAY_USINT[0] := ARRAY_STRUCTURE_AUTO.ARRAY_USINT[0] + 1;
    ARRAY_STRUCTURE_AUTO.ARRAY_USINT[1] := ARRAY_STRUCTURE_AUTO.ARRAY_USINT[1] + 1;
    ARRAY_STRUCTURE_AUTO.ARRAY_USINT[2] := ARRAY_STRUCTURE_AUTO.ARRAY_USINT[2] + 1;
    ARRAY_STRUCTURE_AUTO.ARRAY_USINT[3] := ARRAY_STRUCTURE_AUTO.ARRAY_USINT[3] + 1;
    ARRAY_STRUCTURE_AUTO.ARRAY_USINT[4] := ARRAY_STRUCTURE_AUTO.ARRAY_USINT[4] + 1;
    ARRAY_STRUCTURE_AUTO.ARRAY_USINT[5] := ARRAY_STRUCTURE_AUTO.ARRAY_USINT[5] + 1;
    ARRAY_STRUCTURE_AUTO.ARRAY_USINT[6] := ARRAY_STRUCTURE_AUTO.ARRAY_USINT[6] + 1;
    ARRAY_STRUCTURE_AUTO.ARRAY_USINT[7] := ARRAY_STRUCTURE_AUTO.ARRAY_USINT[7] + 1;
    ARRAY_STRUCTURE_AUTO.ARRAY_USINT[8] := ARRAY_STRUCTURE_AUTO.ARRAY_USINT[6];
    ARRAY_STRUCTURE_AUTO.ARRAY_USINT[9] := ARRAY_STRUCTURE_AUTO.ARRAY_USINT[7];

    ARRAY_STRUCTURE_AUTO.ARRAY_WORD[0] := ARRAY_STRUCTURE_AUTO.ARRAY_WORD[0] + 1;
    ARRAY_STRUCTURE_AUTO.ARRAY_WORD[1] := ARRAY_STRUCTURE_AUTO.ARRAY_WORD[1] + 1;
    ARRAY_STRUCTURE_AUTO.ARRAY_WORD[2] := ARRAY_STRUCTURE_AUTO.ARRAY_WORD[2] + 1;
    ARRAY_STRUCTURE_AUTO.ARRAY_WORD[3] := ARRAY_STRUCTURE_AUTO.ARRAY_WORD[3] + 1;
    ARRAY_STRUCTURE_AUTO.ARRAY_WORD[4] := ARRAY_STRUCTURE_AUTO.ARRAY_WORD[4] + 1;
    ARRAY_STRUCTURE_AUTO.ARRAY_WORD[5] := ARRAY_STRUCTURE_AUTO.ARRAY_WORD[5] + 1;
    ARRAY_STRUCTURE_AUTO.ARRAY_WORD[6] := ARRAY_STRUCTURE_AUTO.ARRAY_WORD[6] + 1;
    ARRAY_STRUCTURE_AUTO.ARRAY_WORD[7] := ARRAY_STRUCTURE_AUTO.ARRAY_WORD[7] + 1;
    ARRAY_STRUCTURE_AUTO.ARRAY_WORD[8] := ARRAY_STRUCTURE_AUTO.ARRAY_WORD[6];
    ARRAY_STRUCTURE_AUTO.ARRAY_WORD[9] := ARRAY_STRUCTURE_AUTO.ARRAY_WORD[7];

END_IF;

END_PROGRAM
